// TIA Portal V18 export
TYPE "SubProcessParameterP010_ShW"
// stored: IsFailsafeCompliant false
   STRUCT
      SubProcessParameter : Struct
         LowerBearingPressingForce : Struct
            LowerBearingPressingForce_value : Real;
            LowerBearingPressingForce_result : Int;
            LowerBearingPressingForce_NG_code : String[9];
         END_STRUCT;
         LowerBearingPressingStroke : Struct
            LowerBearingPressingStroke_value : Real;
            LowerBearingPressingStroke_result : Int;
            LowerBearingPressingStroke_NG_code : String[9];
         END_STRUCT;
         UpperBearingPressingForce : Struct
            UpperBearingPressingForce_value : Real;
            UpperBearingPressingForce_result : Int;
            UpperBearingPressingForce_NG_code : String[9];
         END_STRUCT;
         UpperBearingPressingStroke : Struct
            UpperBearingPressingStroke_value : Real;
            UpperBearingPressingStroke_result : Int;
            UpperBearingPressingStroke_NG_code : String[9];
         END_STRUCT;
         Sleeve1PressingForce : Struct
            Sleeve1PressingForce_value : Real;
            Sleeve1PressingForce_result : Int;
            Sleeve1PressingForce_NG_code : String[9];
         END_STRUCT;
         Sleeve1PressingStroke : Struct
            Sleeve1PressingStroke_value : Real;
            Sleeve1PressingStroke_result : Int;
            Sleeve1PressingStroke_NG_code : String[9];
         END_STRUCT;
         Sleeve2PressingForce : Struct
            Sleeve2PressingForce_value : Real;
            Sleeve2PressingForce_result : Int;
            Sleeve2PressingForce_NG_code : String[9];
         END_STRUCT;
         Sleeve2PressingStroke : Struct
            Sleeve2PressingStroke_value : Real;
            Sleeve2PressingStroke_result : Int;
            Sleeve2PressingStroke_NG_code : String[9];
         END_STRUCT;
      END_STRUCT;
   END_STRUCT;
END_TYPE
